(*
SPDX-FileCopyrightText: © 2026 Oleksandr Tiutyk <trofimich@gmail.com>
SPDX-License-Identifier: MIT
License: https://opensource.org/license/mit
*)

(*!
<summary>
Provides the base lifecycle, state transitions, variable lookup and failure handling for workflow activities.
</summary>
<description>
Activities start from PASSIVE_READY, pause into PASSIVE_SUSPENDED, finish in PASSIVE_COMPLETED,
PASSIVE_HALTED, PASSIVE_CANCELLED or PASSIVE_FAILED, and return to PASSIVE_READY through ACTIVE_RESETTING via
RequestReset. Any uncaught exception in Execute, RequestStart, RequestSuspend, RequestCancel or RequestReset
transitions the activity to PASSIVE_FAILED, copies diagnostics into FailError, invokes OnFail once and
rethrows the exception to the caller. Diagnostic conversion failure stores fixed fallback text. FB_init
stores the workflow association and the default diagnostic name; dynamic instances require
explicit RegisterChild after construction, while static instances remain caller-owned.
PASSIVE_FAILED ends ordinary execution without certifying completion of child or resource cleanup.
Failure handling invokes only synchronous local cleanup. Resource owners must explicitly complete pending
cleanup before sharing or reusing affected resources; resetting may advance that work through OnResetting.
Declared variables reset on successful activity reset, including a reset between loop iterations.
</description>
*)

{attribute 'no_explicit_call' := 'do not call this function block directly'}
FUNCTION_BLOCK ABSTRACT Activity EXTENDS StatefulWorkflowObject
IMPLEMENTS IActivity, ILocalVariableLookup, IVariableResetScopeProvider
VAR
	_Workflow : IWorkflow;

	_ParentActivity : IActivity;

	_VariableResetScope : VariableResetScope;

	_State : WORKFLOW_ELEMENT_STATE;
	_PreviousState : WORKFLOW_ELEMENT_STATE;
	_StateChanged : BOOL;

	_CancelReason : WSTRING(255);
	_HaltReason : WSTRING(255);
END_VAR

(*!
<summary>Reports whether the activity is in an active state requiring cyclic Execute calls.</summary>
<description>
Reports this activity lifecycle only. FALSE does not certify nested resource release after failure.
</description>
*)
{attribute 'monitoring' := 'call'}
PROPERTY FINAL Busy : BOOL
GET
Busy := _State = WORKFLOW_ELEMENT_STATE.ACTIVE_RUNNING
	OR_ELSE _State = WORKFLOW_ELEMENT_STATE.ACTIVE_CANCELLING
	OR_ELSE _State = WORKFLOW_ELEMENT_STATE.ACTIVE_SUSPENDING
	OR_ELSE _State = WORKFLOW_ELEMENT_STATE.ACTIVE_RESETTING;
END_GET
END_PROPERTY

(*!
<summary>Returns the reason recorded for the most recent cancellation request.</summary>
*)
{attribute 'monitoring' := 'call'}
PROPERTY FINAL CancelReason : REFERENCE TO WSTRING(255)
GET
CancelReason REF= _CancelReason;
END_GET
END_PROPERTY

(*!
<summary>Advances the current active state by one step and propagates failures.</summary>
<description>
Dispatches ACTIVE_RUNNING to OnRunning, ACTIVE_CANCELLING and ACTIVE_SUSPENDING to OnStopping, and
ACTIVE_RESETTING to OnResetting. No-op in passive states. When an exception occurs, transitions to
PASSIVE_FAILED, populates FailError, calls OnFail once and rethrows the exception.
</description>
*)
METHOD FINAL Execute
VAR
	runningState : ACTIVITY_RUNNING_STATE;
	stoppingState : ACTIVITY_STOPPING_STATE;
	resettingState : ACTIVITY_RESETTING_STATE;

	haltReason : WSTRING(255);

	exceptionCode : __SYSTEM.ExceptionCode;
END_VAR
_StateChanged := FALSE;

__TRY
	CASE _State OF
		WORKFLOW_ELEMENT_STATE.ACTIVE_RUNNING:
			runningState := OnRunning(startRunning := FALSE, startResuming := FALSE, haltReason => haltReason);

			CASE runningState OF
				ACTIVITY_RUNNING_STATE.WORK_COMPLETED:
					SetNewState(newState := WORKFLOW_ELEMENT_STATE.PASSIVE_COMPLETED);

				ACTIVITY_RUNNING_STATE.WORK_HALTED:
					_HaltReason := haltReason;
					SetNewState(newState := WORKFLOW_ELEMENT_STATE.PASSIVE_HALTED);
			END_CASE

		WORKFLOW_ELEMENT_STATE.ACTIVE_CANCELLING, WORKFLOW_ELEMENT_STATE.ACTIVE_SUSPENDING:
			stoppingState := OnStopping(startCancelling := FALSE, startSuspending := FALSE, haltReason => haltReason);

			CASE stoppingState OF
				ACTIVITY_STOPPING_STATE.WORK_STOPPED:
					IF _State = WORKFLOW_ELEMENT_STATE.ACTIVE_CANCELLING THEN
						SetNewState(newState := WORKFLOW_ELEMENT_STATE.PASSIVE_CANCELLED);
					ELSE
						SetNewState(newState := WORKFLOW_ELEMENT_STATE.PASSIVE_SUSPENDED);
					END_IF

				ACTIVITY_STOPPING_STATE.WORK_COMPLETED:
					SetNewState(newState := WORKFLOW_ELEMENT_STATE.PASSIVE_COMPLETED);

				ACTIVITY_STOPPING_STATE.WORK_HALTED:
					_HaltReason := haltReason;
					SetNewState(newState := WORKFLOW_ELEMENT_STATE.PASSIVE_HALTED);
			END_CASE

		WORKFLOW_ELEMENT_STATE.ACTIVE_RESETTING:
			resettingState := OnResetting(startResetting := FALSE);

			IF resettingState = ACTIVITY_RESETTING_STATE.WORK_RESET THEN
				_FailError.Clear();
				_CancelReason := "";
				_HaltReason := "";
				SetNewState(newState := WORKFLOW_ELEMENT_STATE.PASSIVE_READY);
			END_IF
	END_CASE
__CATCH(exceptionCode)
	handleException(exceptionCode := exceptionCode, catchPointPOUName := __POUNAME(), catchPointPosition := __POSITION());
__ENDTRY
END_METHOD

(*!
<summary>Stores the borrowed workflow association and initializes the default activity name.</summary>
<description>
ClassName must return initialized static storage without reading derived instance fields, raising or
recursively reading Name during base initialization. Does not allocate registry storage. The creator must call
workflow.RegisterChild after __NEW succeeds, outside
lifecycle methods, if the workflow is to own this dynamic instance.
</description>
<param name="workflow">Workflow that hosts this activity. A root requires an explicit association;
0 is allowed for a child that inherits its association from its parent.</param>
*)
METHOD FB_init : BOOL
VAR_INPUT
	bInitRetains : BOOL; // TRUE: the retain variables are initialized (reset warm / reset cold)
	bInCopyCode : BOOL;  // TRUE: the instance will be copied to the copy code afterward (online change)
	workflow : IWorkflow;
END_VAR
_Workflow := workflow;
END_METHOD

(*!
<summary>Borrows the reset scope embedded in this parent for condition attachment.</summary>
<description>Returns live storage for the lifetime of the parent. Used by the validated parent setter
in its owning task. The caller must not delete, copy or independently reconfigure the scope.</description>
*)
METHOD FINAL GetResetScope : IVariableResetScope
GetResetScope := _VariableResetScope;
END_METHOD

(*!
<summary>Returns the diagnostic reason reported when the activity halted its work internally.</summary>
*)
{attribute 'monitoring' := 'call'}
PROPERTY FINAL HaltReason : REFERENCE TO WSTRING(255)
GET
HaltReason REF= _HaltReason;
END_GET
END_PROPERTY

(*!
<summary>
Transitions the activity to PASSIVE_FAILED, records FailError, invokes OnFail and rethrows the exception.
</summary>
<description>
Clones static native exception wrappers before invoking ToError or OnFail so nested exceptions cannot
overwrite the original payload. Conversion failure replaces partial diagnostics with a fixed ERROR fallback;
the original exception is still rethrown. Preserves terminal allocation failure priority before rethrowing.
</description>
<param name="exceptionCode">Caught system exception code.</param>
<param name="catchPointPOUName">Method name where the exception was caught.</param>
<param name="catchPointPosition">Source position where the exception was caught.</param>
*)
METHOD PRIVATE handleException
VAR_INPUT
	exceptionCode : __SYSTEM.ExceptionCode;
	catchPointPOUName : STRING(255);
	catchPointPosition : STRING(255);
END_VAR
VAR
	exception : TOF_Core.IException;
	snapshotAvailable : BOOL;
END_VAR
SetNewState(newState := WORKFLOW_ELEMENT_STATE.PASSIVE_FAILED);

exception := CaptureExecutionException(
	exceptionCode := exceptionCode,
	catchPointPOUName := catchPointPOUName,
	catchPointPosition := catchPointPosition,
	fallbackMessage := "Activity exception diagnostics are unavailable",
	snapshotAvailable => snapshotAvailable
);

__TRY
	OnFail(exception := exception);
__CATCH
__ENDTRY

TOF_Core.DynamicMemoryManager.RaiseIfAllocationFailed();

TOF_Core.ExceptionManager.Throw(exception := exception);
END_METHOD

(*!
<summary>Reports whether variable registration or declaration is blocked by activity or workflow execution.</summary>
*)
METHOD PROTECTED IsVariableScopeBusy : BOOL
VAR
	ownerWorkflow : IWorkflow;
END_VAR
ownerWorkflow := Workflow;

IsVariableScopeBusy := Busy OR_ELSE (ownerWorkflow <> 0 AND_THEN ownerWorkflow.Busy);
END_METHOD

(*!
<summary>Invoked synchronously once when an uncaught exception transitions the activity to PASSIVE_FAILED.</summary>
<description>
Override to perform immediate local stop actions (such as deactivating a timer trigger). Implementations must
not raise exceptions or retain the task-scoped exception reference after returning. Multi-cycle reset work
belongs in OnResetting. Returning from this hook does not certify that pending child or resource operations
have stopped. Keep ownership explicit; a local catch handler cannot infer cleanup completion from this call.
</description>
<param name="exception">Caught exception that caused the failure.</param>
*)
METHOD PROTECTED OnFail
VAR_INPUT
	exception : TOF_Core.IException;
END_VAR
END_METHOD

(*!
<summary>Performs one step of resetting the activity back to PASSIVE_READY.</summary>
<description>
Called with startResetting := TRUE from RequestReset and with startResetting := FALSE on subsequent Execute
calls while in ACTIVE_RESETTING. Return WORK_RESET when internal state, cursors and child activities are ready
for a fresh start, or WORK_IN_PROGRESS when additional Execute cycles are required. The default implementation
returns WORK_RESET immediately.
</description>
<param name="startResetting">TRUE on the initial call from RequestReset; FALSE on cyclic Execute calls.</param>
*)
METHOD PROTECTED OnResetting : ACTIVITY_RESETTING_STATE
VAR_INPUT
	startResetting : BOOL;
END_VAR
OnResetting := ACTIVITY_RESETTING_STATE.WORK_RESET;
END_METHOD

(*!
<summary>Performs one step of activity execution in ACTIVE_RUNNING.</summary>
<description>
Called with startRunning := TRUE on a fresh start from PASSIVE_READY, with startResuming := TRUE when resuming
from PASSIVE_SUSPENDED, and with both flags FALSE on subsequent cyclic Execute calls. Return WORK_IN_PROGRESS
to continue running, WORK_COMPLETED when finished, or WORK_HALTED with haltReason when stopped by internal
logic.
</description>
<param name="startRunning">TRUE on the initial call of a fresh start from PASSIVE_READY.</param>
<param name="startResuming">TRUE on the initial call when resuming from PASSIVE_SUSPENDED.</param>
<param name="haltReason">Diagnostic reason when returning WORK_HALTED.</param>
*)
METHOD PROTECTED ABSTRACT OnRunning : ACTIVITY_RUNNING_STATE
VAR_INPUT
	startRunning : BOOL;
	startResuming : BOOL;
END_VAR
VAR_OUTPUT
	haltReason : WSTRING(255);
END_VAR
END_METHOD

(*!
<summary>Performs one step of cooperative stopping in ACTIVE_CANCELLING or ACTIVE_SUSPENDING.</summary>
<description>
Called with startCancelling := TRUE from RequestCancel, startSuspending := TRUE from RequestSuspend, and with
both flags FALSE on subsequent cyclic Execute calls. Return WORK_IN_PROGRESS while stopping continues,
WORK_STOPPED when the requested cancel or suspend state is reached, WORK_COMPLETED if work completed during
stopping, or WORK_HALTED with haltReason.
</description>
<param name="startCancelling">TRUE on the initial call from RequestCancel.</param>
<param name="startSuspending">TRUE on the initial call from RequestSuspend.</param>
<param name="haltReason">Diagnostic reason when returning WORK_HALTED.</param>
*)
METHOD PROTECTED ABSTRACT OnStopping : ACTIVITY_STOPPING_STATE
VAR_INPUT
	startCancelling : BOOL;
	startSuspending : BOOL;
END_VAR
VAR_OUTPUT
	haltReason : WSTRING(255);
END_VAR
END_METHOD

(*!
<summary>Synchronizes the embedded variable reset scope with the activity variable bindings.</summary>
*)
METHOD PROTECTED OnLocalVariableDeclared
_VariableResetScope.SetBindings(bindings := _VariableScope.Bindings);
END_METHOD

(*!
<summary>Returns the parent workflow element in the hierarchy.</summary>
*)
{attribute 'monitoring' := 'call'}
PROPERTY FINAL Parent : IWorkflowElement
GET
Parent := _ParentActivity;
END_GET
END_PROPERTY

(*!
<summary>Gets or sets the borrowed parent composite activity.</summary>
<description>
An unchanged parent is a no-op. A new parent is validated before mutation; detachment and reparenting are
rejected. Links are borrowed, single-task and stable for the tree lifetime; they do not transfer ownership.
The element, its parent chain and its owning workflow must be PASSIVE_READY during attachment.
</description>
*)
{attribute 'monitoring' := 'call'}
PROPERTY ParentActivity : IActivity
GET
ParentActivity := _ParentActivity;
END_GET
SET
IF _ParentActivity = ParentActivity THEN
	RETURN;
END_IF

IF _ParentActivity <> 0 OR_ELSE ParentActivity = 0 THEN
	WorkflowExceptions.ThrowWorkflowAttachment(
		sourceNamespaceName := NamespaceName,
		sourceClassName := ClassName,
		sourcePOUName := __POUNAME(),
		sourcePosition := __POSITION(),
		message := "Activity parent cannot be detached or replaced"
	);
END_IF

Workflows.ValidateElementAttachment(parent := ParentActivity, child := THIS^);

_ParentActivity := ParentActivity;
END_SET
END_PROPERTY

(*!
<summary>Requests cooperative cancellation of the activity and runs the initial stopping step.</summary>
<description>
No-op when the current state cannot transition to ACTIVE_CANCELLING. Stores the cancellation reason,
transitions to ACTIVE_CANCELLING and invokes OnStopping(TRUE, FALSE). Transitions immediately to
PASSIVE_CANCELLED, PASSIVE_COMPLETED or PASSIVE_HALTED when stopping finishes in one step. On exception,
transitions to PASSIVE_FAILED, populates FailError, calls OnFail and rethrows.
</description>
<param name="reason">Diagnostic reason for cancellation.</param>
*)
METHOD FINAL RequestCancel : BOOL
VAR_INPUT
	reason : WSTRING(255);
END_VAR
VAR
	formattedLogMessage : TOF_Core.ERROR_MESSAGE;

	exceptionCode : __SYSTEM.ExceptionCode;

	stoppingState : ACTIVITY_STOPPING_STATE;
	haltReason : WSTRING(255);
END_VAR
VAR CONSTANT
	targetState : WORKFLOW_ELEMENT_STATE := WORKFLOW_ELEMENT_STATE.ACTIVE_CANCELLING;
END_VAR
formattedLogMessage := TOF_Core.WideStrings.Concat255("Cancel requested for activity '", Name, "'");

TOF_Core.LogManager.TryLogMessage(
	message := formattedLogMessage,
	category := TOF_Core.LOG_CATEGORY.INFORMATION,
	topic1 := "Activity",
	topic2 := "ActivityRequest",
	topic3 := "ActivityRequestCancel"
);

IF NOT Workflows.ValidateTransition(currentState := _State, newState := targetState) THEN
	RequestCancel := FALSE;
	RETURN;
END_IF

SetNewState(newState := targetState);
_CancelReason := reason;

__TRY
	stoppingState := OnStopping(startCancelling := TRUE, startSuspending := FALSE, haltReason => haltReason);

	CASE stoppingState OF
		ACTIVITY_STOPPING_STATE.WORK_STOPPED:
			SetNewState(newState := WORKFLOW_ELEMENT_STATE.PASSIVE_CANCELLED);

		ACTIVITY_STOPPING_STATE.WORK_COMPLETED:
			SetNewState(newState := WORKFLOW_ELEMENT_STATE.PASSIVE_COMPLETED);

		ACTIVITY_STOPPING_STATE.WORK_HALTED:
			_HaltReason := haltReason;
			SetNewState(newState := WORKFLOW_ELEMENT_STATE.PASSIVE_HALTED);
	END_CASE
__CATCH(exceptionCode)
	handleException(exceptionCode := exceptionCode, catchPointPOUName := __POUNAME(), catchPointPosition := __POSITION());
__ENDTRY

RequestCancel := TRUE;
END_METHOD

(*!
<summary>Requests resetting from a finished passive state and runs the initial resetting step.</summary>
<description>
Permitted from PASSIVE_COMPLETED, PASSIVE_HALTED, PASSIVE_CANCELLED and PASSIVE_FAILED; no-op in other states.
Transitions to ACTIVE_RESETTING and invokes OnResetting(startResetting := TRUE). When WORK_RESET is returned immediately, clears
FailError, CancelReason and HaltReason and transitions to PASSIVE_READY in the same call. On exception,
transitions to PASSIVE_FAILED, populates FailError, calls OnFail and rethrows.
</description>
*)
METHOD FINAL RequestReset : BOOL
VAR
	formattedLogMessage : TOF_Core.ERROR_MESSAGE;

	exceptionCode : __SYSTEM.ExceptionCode;
	resettingState : ACTIVITY_RESETTING_STATE;
END_VAR
VAR CONSTANT
	targetState : WORKFLOW_ELEMENT_STATE := WORKFLOW_ELEMENT_STATE.ACTIVE_RESETTING;
END_VAR
formattedLogMessage := TOF_Core.WideStrings.Concat255("Reset requested for activity '", Name, "'");

TOF_Core.LogManager.TryLogMessage(
	message := formattedLogMessage,
	category := TOF_Core.LOG_CATEGORY.INFORMATION,
	topic1 := "Activity",
	topic2 := "ActivityRequest",
	topic3 := "ActivityRequestReset"
);

IF NOT Workflows.ValidateTransition(currentState := _State, newState := targetState) THEN
	RequestReset := FALSE;
	RETURN;
END_IF

SetNewState(newState := targetState);

__TRY
	resettingState := OnResetting(startResetting := TRUE);

	IF resettingState = ACTIVITY_RESETTING_STATE.WORK_RESET THEN
		_FailError.Clear();
		_CancelReason := "";
		_HaltReason := "";
		SetNewState(newState := WORKFLOW_ELEMENT_STATE.PASSIVE_READY);
	END_IF
__CATCH(exceptionCode)
	handleException(exceptionCode := exceptionCode, catchPointPOUName := __POUNAME(), catchPointPosition := __POSITION());
__ENDTRY

RequestReset := TRUE;
END_METHOD

(*!
<summary>
Requests a fresh start from PASSIVE_READY or resumes from PASSIVE_SUSPENDED and runs the initial step.
</summary>
<description>
No-op when the current state cannot transition to ACTIVE_RUNNING. Clears prior run diagnostics, transitions to
ACTIVE_RUNNING and invokes OnRunning. Transitions immediately to PASSIVE_COMPLETED or PASSIVE_HALTED if
finished in one step. On exception, transitions to PASSIVE_FAILED, populates FailError, calls OnFail and
rethrows.
</description>
*)
METHOD FINAL RequestStart : BOOL
VAR
	formattedLogMessage : TOF_Core.ERROR_MESSAGE;

	resuming : BOOL;

	exceptionCode : __SYSTEM.ExceptionCode;

	runningState : ACTIVITY_RUNNING_STATE;
	haltReason : WSTRING(255);
END_VAR
VAR CONSTANT
	targetState : WORKFLOW_ELEMENT_STATE := WORKFLOW_ELEMENT_STATE.ACTIVE_RUNNING;
END_VAR
formattedLogMessage := TOF_Core.WideStrings.Concat255("Start requested for activity '", Name, "'");

TOF_Core.LogManager.TryLogMessage(
	message := formattedLogMessage,
	category := TOF_Core.LOG_CATEGORY.INFORMATION,
	topic1 := "Activity",
	topic2 := "ActivityRequest",
	topic3 := "ActivityRequestStart"
);

IF NOT Workflows.ValidateTransition(currentState := _State, newState := targetState) THEN
	RETURN;
END_IF

resuming := _State = WORKFLOW_ELEMENT_STATE.PASSIVE_SUSPENDED;

SetNewState(newState := targetState);

_FailError.Clear();
_CancelReason := "";
_HaltReason := "";

__TRY
	runningState := OnRunning(startRunning := NOT resuming, startResuming := resuming, haltReason => haltReason);

	CASE runningState OF
		ACTIVITY_RUNNING_STATE.WORK_COMPLETED:
			SetNewState(newState := WORKFLOW_ELEMENT_STATE.PASSIVE_COMPLETED);

		ACTIVITY_RUNNING_STATE.WORK_HALTED:
			_HaltReason := haltReason;
			SetNewState(newState := WORKFLOW_ELEMENT_STATE.PASSIVE_HALTED);
	END_CASE
__CATCH(exceptionCode)
	handleException(exceptionCode := exceptionCode, catchPointPOUName := __POUNAME(), catchPointPosition := __POSITION());
__ENDTRY

RequestStart := TRUE;
END_METHOD

(*!
<summary>Requests cooperative suspension from ACTIVE_RUNNING and runs the initial stopping step.</summary>
<description>
No-op when the current state cannot transition to ACTIVE_SUSPENDING. Transitions to ACTIVE_SUSPENDING and
invokes OnStopping(FALSE, TRUE). Transitions immediately to PASSIVE_SUSPENDED, PASSIVE_COMPLETED or
PASSIVE_HALTED if stopping finishes in one step. On exception, transitions to PASSIVE_FAILED, populates
FailError, calls OnFail and rethrows.
</description>
*)
METHOD FINAL RequestSuspend : BOOL
VAR
	formattedLogMessage : TOF_Core.ERROR_MESSAGE;

	exceptionCode : __SYSTEM.ExceptionCode;

	stoppingState : ACTIVITY_STOPPING_STATE;
	haltReason : WSTRING(255);
END_VAR
VAR CONSTANT
	targetState : WORKFLOW_ELEMENT_STATE := WORKFLOW_ELEMENT_STATE.ACTIVE_SUSPENDING;
END_VAR
formattedLogMessage := TOF_Core.WideStrings.Concat255("Suspend requested for activity '", Name, "'");

TOF_Core.LogManager.TryLogMessage(
	message := formattedLogMessage,
	category := TOF_Core.LOG_CATEGORY.INFORMATION,
	topic1 := "Activity",
	topic2 := "ActivityRequest",
	topic3 := "ActivityRequestSuspend"
);

IF NOT Workflows.ValidateTransition(currentState := _State, newState := targetState) THEN
	RequestSuspend := FALSE;
	RETURN;
END_IF

SetNewState(newState := targetState);

__TRY
	stoppingState := OnStopping(startCancelling := FALSE, startSuspending := TRUE, haltReason => haltReason);

	CASE stoppingState OF
		ACTIVITY_STOPPING_STATE.WORK_STOPPED:
			SetNewState(newState := WORKFLOW_ELEMENT_STATE.PASSIVE_SUSPENDED);

		ACTIVITY_STOPPING_STATE.WORK_COMPLETED:
			SetNewState(newState := WORKFLOW_ELEMENT_STATE.PASSIVE_COMPLETED);

		ACTIVITY_STOPPING_STATE.WORK_HALTED:
			_HaltReason := haltReason;
			SetNewState(newState := WORKFLOW_ELEMENT_STATE.PASSIVE_HALTED);
	END_CASE
__CATCH(exceptionCode)
	handleException(exceptionCode := exceptionCode, catchPointPOUName := __POUNAME(), catchPointPosition := __POSITION());
__ENDTRY

RequestSuspend := TRUE;
END_METHOD

(*!
<summary>Updates the activity state, records the transition flag and logs the state change.</summary>
<description>
No-op when newState equals the current state. Successful reset restores local and attached condition declarations.
</description>
<param name="newState">New workflow element state to assign.</param>
*)
METHOD PROTECTED FINAL SetNewState
VAR_INPUT
	newState : WORKFLOW_ELEMENT_STATE;
END_VAR
VAR
	formattedLogMessage : TOF_Core.ERROR_MESSAGE;
END_VAR
IF _State = newState THEN
	RETURN;
END_IF

formattedLogMessage := TOF_Core.WideStrings.Concat255(
	"Activity '",
	Name,
	"' state changed from '",
	TO_WSTRING(_State),
	"' to '",
	TO_WSTRING(newState),
	"'"
);

TOF_Core.LogManager.TryLogMessage(
	message := formattedLogMessage,
	category := TOF_Core.LOG_CATEGORY.INFORMATION,
	topic1 := "Activity",
	topic2 := "ActivitySetNewState"
);

IF _State = WORKFLOW_ELEMENT_STATE.ACTIVE_RESETTING AND_THEN newState = WORKFLOW_ELEMENT_STATE.PASSIVE_READY THEN
	_VariableResetScope.Restore();
END_IF

_PreviousState := _State;
_State := newState;
_StateChanged := TRUE;
END_METHOD

(*!
<summary>Returns the current lifecycle state of the activity.</summary>
*)
{attribute 'monitoring' := 'call'}
PROPERTY FINAL State : WORKFLOW_ELEMENT_STATE
GET
State := _State;
END_GET
END_PROPERTY

(*!
<summary>Attempts to find a binding registered directly on this instance.</summary>
<description>
Does not inspect parents or workflow fallback. Returns a borrowed descriptor only on TRUE.
Returns FALSE for absence, callback exceptions or terminal allocation failure without clearing the fatal latch.
The owner keeps the registered PLC storage alive; use one task without concurrent reconfiguration.
</description>
<param name="name">Case-sensitive name registered directly on this instance.</param>
<param name="variable">Borrowed binding descriptor, usable only on TRUE.</param>
*)
METHOD TryGetLocalVariable : BOOL
VAR_INPUT
	name : STRING;
END_VAR
VAR_OUTPUT
	variable : TOF_Core.GENERIC_VALUE;
END_VAR
TryGetLocalVariable := _VariableScope.TryGetLocalVariable(name := name, variable => variable);
END_METHOD

(*!
<summary>Attempts to resolve a named variable from this activity, its ancestor activities or the workflow.</summary>
<description>
Returns FALSE when resolution fails or a nested call raises an exception. Use the output only when TRUE is
returned. Does not propagate exceptions or clear terminal allocation state. A latched allocation failure returns FALSE
without entering further lookup callbacks, including when a nested callback contained the allocation exception.
</description>
<param name="name">Case-sensitive variable name to look up.</param>
<param name="variable">Resolved variable value when TRUE is returned.</param>
*)
METHOD TryGetVariable : BOOL
VAR_INPUT
	name : STRING;
END_VAR
VAR_OUTPUT
	variable : TOF_Core.GENERIC_VALUE;
END_VAR
IF TOF_Core.DynamicMemoryManager.HasAllocationFailed THEN
	RETURN;
END_IF

__TRY
	TryGetVariable := _VariableScope.TryGetLocalVariable(name := name, variable => variable);

	IF NOT TryGetVariable AND_THEN NOT TOF_Core.DynamicMemoryManager.HasAllocationFailed
		AND_THEN _ParentActivity <> 0
	THEN
		TryGetVariable := _ParentActivity.TryGetVariable(name := name, variable => variable);
	END_IF

	IF NOT TryGetVariable AND_THEN NOT TOF_Core.DynamicMemoryManager.HasAllocationFailed
		AND_THEN _Workflow <> 0
	THEN
		TryGetVariable := _Workflow.TryGetVariable(name := name, variable => variable);
	END_IF
__CATCH
	TryGetVariable := FALSE;
__ENDTRY

IF TOF_Core.DynamicMemoryManager.HasAllocationFailed THEN
	TryGetVariable := FALSE;
END_IF
END_METHOD

(*!
<summary>Returns the diagnostic owner kind label ('activity') for variable registration errors.</summary>
*)
METHOD PROTECTED VariableScopeOwnerKind : STRING
VariableScopeOwnerKind := 'activity';
END_METHOD

(*!
<summary>Returns the workflow associated with this activity or inherited from its parent activity.</summary>
*)
{attribute 'monitoring' := 'call'}
PROPERTY Workflow : IWorkflow
GET
IF _Workflow <> 0 THEN
	Workflow := _Workflow;
ELSIF _ParentActivity <> 0 THEN
	Workflow := _ParentActivity.Workflow;
END_IF
END_GET
END_PROPERTY

(*!
<summary>Indicates whether RequestCancel is permitted in the current activity state.</summary>
*)
{attribute 'monitoring' := 'call'}
{attribute 'OPC.UA.DA.Property' := '1'}
{attribute 'OPC.UA.DA.Access' := '1'}
PROPERTY FINAL CancellingAllowed : BOOL
GET
CancellingAllowed := Workflows.ValidateTransition(
	currentState := _State,
	newState := WORKFLOW_ELEMENT_STATE.ACTIVE_CANCELLING
);
END_GET
END_PROPERTY

(*!
<summary>Indicates whether RequestReset is permitted in the current activity state.</summary>
*)
{attribute 'monitoring' := 'call'}
{attribute 'OPC.UA.DA.Property' := '1'}
{attribute 'OPC.UA.DA.Access' := '1'}
PROPERTY FINAL ResettingAllowed : BOOL
GET
ResettingAllowed := Workflows.ValidateTransition(
	currentState := _State,
	newState := WORKFLOW_ELEMENT_STATE.ACTIVE_RESETTING
);
END_GET
END_PROPERTY

(*!
<summary>Indicates whether RequestStart is permitted in the current activity state.</summary>
*)
{attribute 'monitoring' := 'call'}
{attribute 'OPC.UA.DA.Property' := '1'}
{attribute 'OPC.UA.DA.Access' := '1'}
PROPERTY FINAL StartingAllowed : BOOL
GET
StartingAllowed := Workflows.ValidateTransition(
	currentState := _State,
	newState := WORKFLOW_ELEMENT_STATE.ACTIVE_RUNNING
);
END_GET
END_PROPERTY

(*!
<summary>Indicates whether RequestSuspend is permitted in the current activity state.</summary>
*)
{attribute 'monitoring' := 'call'}
{attribute 'OPC.UA.DA.Property' := '1'}
{attribute 'OPC.UA.DA.Access' := '1'}
PROPERTY FINAL SuspendingAllowed : BOOL
GET
SuspendingAllowed := Workflows.ValidateTransition(
	currentState := _State,
	newState := WORKFLOW_ELEMENT_STATE.ACTIVE_SUSPENDING
);
END_GET
END_PROPERTY

END_FUNCTION_BLOCK

(* stored: Version 1.1.0.1
   POU Activity: Id {ab48bd8b-e561-4a48-ba30-d8d6aa6a3a44}, SpecialFunc None
   Folder Methods to override: Id {e7dec774-a925-4c60-82fb-0de6b314c0cf}
   Folder Overriden methods: Id {62d4e78a-f501-447a-9a03-7cb7d189b2ce}
   Folder Service methods: Id {d209e4cb-f636-4994-9756-8ec05d532d51}
   Property Busy: Id {4a27e4a6-049e-423b-bd5e-9b17f40d26c7}
   Get Get: Id {051f0622-8617-4132-bb68-a981920bece1}
   Property CancelReason: Id {e2bc3f04-4677-4d3c-9357-f54296f5e5c8}
   Get Get: Id {df206a6b-d527-4e14-aba8-68798b8c9d03}
   Method Execute: Id {be6fc6c1-8eae-4046-84ea-8d4eaff4bdc8}
   Method FB_init: Id {ffd89157-0584-4da6-8b2f-193481b5613d}
   Method GetResetScope: Id {f95f8a74-1574-438b-999e-7247a44ca556}
   Property HaltReason: Id {07437ef7-469f-4431-94a0-8d23aebd0d97}
   Get Get: Id {f06593a6-8dcc-4d84-a248-9dce2650988b}
   Method handleException: Id {a2f46e54-8b11-4431-a8d7-849983a96601}
   Method IsVariableScopeBusy: Id {91e4b308-5d27-4a69-8f13-2c70d48e6b54}
   Method OnFail: Id {86d98c43-34b6-41e3-a2de-bfa6e2663324}
   Method OnResetting: Id {d4c17a91-67e5-4d91-9e12-54c3b886e712}
   Method OnRunning: Id {ff3568b9-81d7-45c0-aad6-1ecbde24ba04}
   Method OnStopping: Id {0f732c8a-9e9a-4779-80c6-a3e254a4c94f}
   Method OnLocalVariableDeclared: Id {4c82d109-6f35-4b81-a927-3e50c48f7d62}
   Property Parent: Id {d42ed62d-e5ae-493d-a21e-c03f60e3c88f}
   Get Get: Id {765fc5b2-4f23-4c68-98f4-2352c4c6e3f2}
   Property ParentActivity: Id {7746eee7-81b2-4cc8-b04b-86aaff99c3e3}
   Get Get: Id {c910d929-401b-4d62-9e02-b489beb98812}
   Set Set: Id {45312744-e8d0-4156-ae50-a2d68cc6dcc8}
   Method RequestCancel: Id {b3ceac03-f171-4dc0-9de1-bd85e0183af2}
   Method RequestReset: Id {b882054b-41a4-4a62-9946-6bd084653f81}
   Method RequestStart: Id {09722d60-5a50-4ba0-834d-aa751d69d95a}
   Method RequestSuspend: Id {2ed6294f-7e81-48bb-96fc-22593c00015d}
   Method SetNewState: Id {7af2da96-4196-4a37-93e6-687784f94a02}
   Property State: Id {201c6b82-3a53-42a5-a4be-54bc270d67ef}
   Get Get: Id {a6a927b4-af82-407a-901f-2a288505a083}
   Method TryGetLocalVariable: Id {94a358d5-d57f-4692-8c09-8e852ed362d3}
   Method TryGetVariable: Id {7404742e-521b-4644-b536-622820cce67b}
   Method VariableScopeOwnerKind: Id {7d28f419-3e65-4b82-9a14-6c50d27e8f31}
   Property Workflow: Id {5b9f0838-cfd8-4e68-96b0-62c7d023998f}
   Get Get: Id {82ce28f2-8424-4b0f-9ba1-3ba80b3f14e7}
   Property CancellingAllowed: Id {868305a0-a5de-4fb8-b3cf-2cf01059ea30}
   Get Get: Id {b12c0fe2-db0a-4997-b709-e758605575c6}
   Property ResettingAllowed: Id {49b974b3-692b-4212-8638-6ed8ee337c3a}
   Get Get: Id {bacbd5e5-a6b8-49ad-b6e5-2270b29684d9}
   Property StartingAllowed: Id {0e57024a-4369-4bb0-bb72-733b9c164be7}
   Get Get: Id {f58b9199-dadb-410f-af91-1aae549d7681}
   Property SuspendingAllowed: Id {792c5c33-41f1-4ff2-9a1a-465498db704c}
   Get Get: Id {df911083-c53c-490b-a5da-ff5e491736f8} *)
